# EPICS IOC start-up script: test/startup/st.mcu007-Dct-streamdevice.iocsh
#require EthercatMC,USER

epicsEnvSet("MOTOR_PORT",    "$(SM_MOTOR_PORT=MCU1)")

epicsEnvSet("IPADDR",        "$(SM_IPADDR=172.30.244.150)")
epicsEnvSet("IPPORT",        "$(SM_IPPORT=5000)")
epicsEnvSet("ASYN_PORT",     "$(SM_ASYN_PORT=MC_CPU1)")
epicsEnvSet("PREFIX",        "$(SM_PREFIX=LabS-MCAG:MC-MCU-07:)")
epicsEnvSet("STREAM_PROTOCOL_PATH", "db")

epicsEnvSet("PREC",          "$(SM_PREC=3)")

< ethercatmcDctEL1252-Stream.iocsh
